{attribute addProperty BoxType "EL3101-0000-0016"}
{attribute addProperty Id "StatusAT %I*Status_F9B4A0131621ValueAT %I*INT16217"}
{attribute addProperty CRC "2420590242"}
{attribute addProperty SizeInBites "32"}
{attribute addProperty SizeInBytes "4"}
TYPE AI_Standard_904746A2 :
STRUCT
	{attribute addProperty Name "Status"}
	Status AT %I* : Status_F9B4A013;
	{attribute addProperty Name "Value"}
	Value AT %I* : INT;
END_STRUCT
END_TYPE

(* stored: Version 1.2.0.0, ProductVersion 3.1.4024.9
   DUT AI_Standard_904746A2: Id {ce6a22dd-91a5-4eeb-9f2f-048f7225be1f} *)
